Staubli VAL3: Day7.dtx

string sInput
num nInput
lists lResult
  [0]
    string sString
num nResult
num nInput2
num nCounter[9]
num nResult2
num nInput1
num nMedian
num nDiff
num nRange
num nSum
num nDiffGuess
num nFuel
